Staubli VAL3: onF1Event.pgx

program onF1Event()
  local num i
  local string l_sItem
begin
  // load the page AXIS7

end
